PROGRAM main
VAR
    kitchen     : Kitchen;
    dining_room : Room;
    living_room : Room;
    bedroom     : ARRAY [0..(house.N_BEDROOMS-1)]  OF Room;
    bathroom    : ARRAY [0..(house.N_BATHROOMS-1)] OF Room;

    i           : USINT := 0;
END_VAR

kitchen(target_luminosity_lumens := 1300, target_temperature_oc := 19.5, n_broccolis := 3);
dining_room(target_luminosity_lumens := 1100, target_temperature_oc := 19.5);
living_room(target_luminosity_lumens := 800, target_temperature_oc := 19.5);

FOR i := 0 TO (house.N_BEDROOMS-1) DO
    bedroom[i](target_luminosity_lumens := 600, target_temperature_oc := 16.0);
END_FOR

FOR i := 0 TO (house.N_BATHROOMS-1) DO
    bathroom[i](target_luminosity_lumens := 1300, target_temperature_oc := 18.5);
END_FOR

END_PROGRAM

(* stored: Version 1.1.0.1, ProductVersion 3.1.4024.13
   POU main: Id {203fc978-33c9-4170-91a9-66c47706bd0f}, SpecialFunc None *)
